Yaskawa INFORM job: CODER.JBI

/JOB
//NAME MOV_TY
//POS
///NPOS 2,2,0,0
///TOOL 2
///RECTAN
///RCONF 0,0,0,0,0
C000=920.760,-872.449,765.394,-30.30,88.06,-118.61
C001=920.760,-872.426,765.391,-177.26,68.98,94.24
E000=-0.367,,,,,
E001=-0.367,,,,,
//INST
///DATE 2010/05/04 13:42
///ATTR 0,0,0,0,0,0,0,0,0,0,0,0,1,0,0,0
///FRAME 1
NOP
MOVL C000 E000 V=0.1 CONT
MOVL C001 E001 V=0.1 CONT
END
